FUNCTION_BLOCK FB_Valve_0_10V IMPLEMENTS I_Valve
VAR_INPUT
END_VAR
VAR_OUTPUT
END_VAR
VAR
		//Properties
	bError : BOOL := FALSE;
	fOpeningActual : REAL;
	fOpeningSetpoint : REAL := 0;
	//Raw values
	nOpeningSet AT %Q* : INT;
	nOpeningAct AT %I* : INT;
END_VAR

{warning 'Eigenschaftenimplementierung hinzufügen'}
PROPERTY Error : BOOL
GET
Error := THIS^.bError;
END_GET
SET
THIS^.bError := Error;
END_SET
END_PROPERTY

{warning 'Eigenschaftenimplementierung hinzufügen'}
PROPERTY OpeningActual : REAL
GET
OpeningActual := THIS^.fOpeningActual;
END_GET
SET
THIS^.fOpeningActual := OpeningActual;
END_SET
END_PROPERTY

{warning 'Eigenschaftenimplementierung hinzufügen'}
PROPERTY OpeningSetpoint : REAL
GET
OpeningSetpoint := THIS^.fOpeningSetpoint;
END_GET
SET
THIS^.fOpeningSetpoint := OpeningSetpoint;
END_SET
END_PROPERTY

{warning 'Methodenimplementierung hinzufügen'}
METHOD Run
//Read feedback for opening position
fOpeningActual := FC_Voltage0_10Raw_TO_Percentage(nOpeningAct);

//Write setpoint for opening position
nOpeningSet := FC_Percentage_TO_Voltage0_10Raw(fOpeningSetpoint);
END_METHOD

END_FUNCTION_BLOCK

(* stored: Version 1.1.0.1, ProductVersion 3.1.4024.3
   POU FB_Valve_0_10V: Id {1e12148b-6fe4-4147-8e61-fbd5c548397a}, SpecialFunc None
   Property Error: Id {2fed5cb7-e454-4e37-8408-6f50394c5994}
   Get Get: Id {27aff8c1-86ec-4cf2-b6ca-d0f91c1153dd}
   Set Set: Id {90539a20-3ee7-40c1-8025-084bf51c696a}
   Property OpeningActual: Id {e6bcae82-10a5-4eb7-a50c-69eb697d2e4e}
   Get Get: Id {57218f8f-c451-492f-92ac-205af2d952b0}
   Set Set: Id {b28651fa-d17d-4be8-a0e7-7daf35ea411a}
   Property OpeningSetpoint: Id {7646cfd6-c0a4-408b-9d4e-2b2eae0d8ef1}
   Get Get: Id {f304f1c1-d23b-45de-b1d6-ce2625ccbe72}
   Set Set: Id {fae38abd-5d53-43a9-ad6b-25320fa19904}
   Method Run: Id {e66636cb-76a0-483f-9013-19ae960a28da} *)
